// SIMATIC STEP 7 (V5.x) project S_M_Desbobinado
// CPU: CPU312(1)
// station: P_ADR_BUS
// station: Hardware
// station: Equipo SIMATIC 300
// program: Programa S7(1)

SYMBOL_TABLE
"CONTADOR"	C 1	COUNTER
"DESBOBINADO"	FB 1	FB 1	// Función que se encarga del desbobinado
"MULT"	FB 2	FB 2
"MULT_DEBOB"	FB 3	FB 3
"S_CACEROLA"	I 124.0	BOOL
"S_SARTEN"	I 124.1	BOOL
"S_PAELLERA"	I 124.2	BOOL
"S_WOK"	I 124.3	BOOL
"PRESENCIA"	I 124.4	BOOL
"BIT_DE_TRABAJO"	I 124.5	BOOL
"START"	I 124.6	BOOL
"BAJAR_CONT"	I 124.7	BOOL
"SARTEN"	I 125.0	BOOL
"CACEROLA"	I 125.1	BOOL
"WOK"	I 125.2	BOOL
"PAELLERA"	I 125.3	BOOL
"Cycle Execution"	OB 1	OB 1
"C_CACEROLA"	PIW 651	INT
"C_SARTEN"	PIW 653	INT
"C_WOK"	PIW 655	INT
"C_PAELLERA"	PIW 657	INT
"MCENTRO"	PIW 659	INT
"PLANCHAS"	PIW 661	WORD
"ABRIRMCENTRO"	Q 100.0	BOOL
"DESBOBINAR"	Q 100.1	BOOL
"BIT_OK"	Q 100.2	BOOL
"BIT_ERROR"	Q 100.3	BOOL
"STBY"	Q 100.4	BOOL
"STBY_SARTEN"	Q 101.0	BOOL
"STBY_CACEROLA"	Q 101.1	BOOL
"STBY_PAELLERA"	Q 101.2	BOOL
"STBY_WOK"	Q 101.3	BOOL
END_SYMBOL_TABLE

FUNCTION_BLOCK "DESBOBINADO"	// FB 1
TITLE = DESBOBINADO
VERSION : 0.1
VAR_INPUT
  SENSOR : BOOL ;
  PRESENCIA : BOOL ;
  CENTRO : INT ;
  bit_de_trabajo : BOOL ;
  MCENTRO : INT ;
  Contador : COUNTER ;
  START : BOOL ;
  PLANCHAS : WORD  := W#16#100;
END_VAR
VAR_OUTPUT
  ABRIRMCENTRO : BOOL ;
  DESBOBINAR : BOOL ;
  STBY : BOOL ;
END_VAR
VAR
  x31 : BOOL ;
  x32 : BOOL ;
  x33 : BOOL ;
  x34 : BOOL ;
  s1 : BOOL ;
  FP_Bit_Tr : BOOL ;
  x30 : BOOL ;
  FP_PRESENCIA : BOOL ;
  FP_BDT : BOOL ;
  FP_START : BOOL ;
END_VAR
VAR_TEMP
  watchdog_master : BOOL ;
END_VAR
BEGIN
NETWORK
TITLE = Arranque
      SET;
      A     #bit_de_trabajo;
      FP    #FP_BDT;
      S     #x30;
      R     #x31;
      R     #x32;
      R     #x33;
      R     #x34;
      R     #s1;
NETWORK
TITLE = x31 a x32
//Comparacion medida centro con medida nominal del centro para pasar de x31 a x32
      A     #x31;
      A(;
      L     #CENTRO;
      L     #MCENTRO;
      ==R;
      );
      R     #x31;
      S     #x32;
NETWORK
TITLE = x32 a x33
//Presencia detecta que la plancha esta en posicion para empezar el proceso de 
//desbobinado-cizallado
      A     #x32;
      A     #PRESENCIA;
      FP    #FP_PRESENCIA;
      R     #x32;
      S     #x33;
NETWORK
TITLE = x33 a x34
//Detecta que la plancha esta lista para ser cizallada
      A     #x33;
      A     #SENSOR;
      R     #x33;
      S     #x34;
NETWORK
TITLE = x34 a x33
//si el contador no ha acabado
      A     #x34;
      T     LD 1;
      TAK;
      T     LD 5;
      L     #Contador;
      T     LW 9;
      L     LD 5;
      L     LD 1;
      A     C [LW 9];
      AN    #SENSOR;
      R     #x34;
      S     #x33;
NETWORK
TITLE = x34 a s1
//si el contador ha cabado
      A     #x34;
      T     LD 1;
      TAK;
      T     LD 5;
      L     #Contador;
      T     LW 9;
      L     LD 5;
      L     LD 1;
      AN    C [LW 9];
      AN    #SENSOR;
      AN    #PRESENCIA;
      R     #x34;
      S     #x30;
NETWORK
TITLE = Tratamiento de bit de fin
      A     #x30;
      =     #STBY;
NETWORK
TITLE = Abrir centro
      A     #x31;
      =     #ABRIRMCENTRO;
NETWORK
TITLE = Carga del contador y desbobinado en x32
      A     #x32;
      S     #DESBOBINAR;
      L     #PLANCHAS;
      T     LD 1;
      TAK;
      T     LD 5;
      L     #Contador;
      T     LW 9;
      L     LD 5;
      L     LD 1;
      S     C [LW 9];
NETWORK
TITLE = Resta del contador y salida del x33
      A     #x33;
      S     #DESBOBINAR;
NETWORK
TITLE =
      A     #x34;
      R     #DESBOBINAR;
NETWORK
TITLE = De X30 a X31
      A     #START;
      FP    #FP_START;
      A     #x30;
      R     #x30;
      S     #x31;
END_FUNCTION_BLOCK

FUNCTION_BLOCK "MULT_DEBOB"	// FB 3
VERSION : 0.1
VAR_INPUT
  S_CACEROLA : BOOL ;
  S_SARTEN : BOOL ;
  S_PAELLERA : BOOL ;
  S_WOK : BOOL ;
  PRESENCIA : BOOL ;
  C_CACEROLA : INT ;
  C_SARTEN : INT ;
  C_WOK : INT ;
  C_PAELLERA : INT ;
  BIT_DE_TRABAJO : BOOL ;
  MCENTRO : INT ;
  CONTADOR : COUNTER ;
  PLANCHAS : WORD ;
  SARTEN : BOOL ;
  CACEROLA : BOOL ;
  WOK : BOOL ;
  PAELLERA : BOOL ;
  START : BOOL ;
END_VAR
VAR_OUTPUT
  ABRIRMCENTRO : BOOL ;
  DESBOBINAR : BOOL ;
  BIT_OK : BOOL ;
  BIT_ERROR : BOOL ;
  STBY : BOOL ;
  STBY_SAR : BOOL ;
  STBY_CAC : BOOL ;
  STBY_WOK : BOOL ;
  STBY_PAELL : BOOL ;
END_VAR
VAR
  CAC_DESB : FB 1;
  SART_DESB : FB 1;
  WOK_DESB : FB 1;
  PAELL_DESB : FB 1;
  START_SAR : BOOL ;
  START_CAC : BOOL ;
  START_WOK : BOOL ;
  START_PAELL : BOOL ;
  FP_BDT : BOOL ;
  X1 : BOOL ;
  X2 : BOOL ;
  X3 : BOOL ;
  X4 : BOOL ;
  X5 : BOOL ;
  X6 : BOOL ;
  BDT : BOOL ;
  FP_START : BOOL ;
  FLAG_DESB : BOOL ;
  FP_DESBOB : BOOL ;
  F_START : BOOL ;
END_VAR
BEGIN
NETWORK
TITLE =
      A     #X2;
      JCN   _008;
      S     #BDT;
      BLD   14;
      =     L 6.0;
      L     DINO;
      T     LW 4;
      CDB;
      OPN   DI [LW 4];
      TAR2  LD 0;
      A     DBX [AR2,P#0.1];
      =     #SART_DESB.SENSOR;
      A     DBX [AR2,P#0.4];
      =     #SART_DESB.PRESENCIA;
      L     DBW [AR2,P#4.0];
      T     #SART_DESB.CENTRO;
      A     DBX [AR2,P#95.3];
      =     #SART_DESB.bit_de_trabajo;
      L     DBW [AR2,P#12.0];
      T     #SART_DESB.MCENTRO;
      L     DBW [AR2,P#14.0];
      T     #SART_DESB.Contador;
      A     DBX [AR2,P#94.0];
      =     #SART_DESB.START;
      L     DBW [AR2,P#16.0];
      T     #SART_DESB.PLANCHAS;
      +AR2  P#40.0;
      UC    "DESBOBINADO";
      LAR2  LD 0;
      A     #SART_DESB.ABRIRMCENTRO;
      =     DBX [AR2,P#20.0];
      A     #SART_DESB.DESBOBINAR;
      =     DBX [AR2,P#20.1];
      A     #SART_DESB.STBY;
      =     DBX [AR2,P#20.5];
      CDB;
      BLD   15;
_008: NOP   0;
NETWORK
TITLE =
      A     #X3;
      JCN   _009;
      S     #BDT;
      BLD   14;
      =     L 6.0;
      L     DINO;
      T     LW 4;
      CDB;
      OPN   DI [LW 4];
      TAR2  LD 0;
      A     DBX [AR2,P#0.0];
      =     #CAC_DESB.SENSOR;
      A     DBX [AR2,P#0.4];
      =     #CAC_DESB.PRESENCIA;
      L     DBW [AR2,P#2.0];
      T     #CAC_DESB.CENTRO;
      A     DBX [AR2,P#95.3];
      =     #CAC_DESB.bit_de_trabajo;
      L     DBW [AR2,P#12.0];
      T     #CAC_DESB.MCENTRO;
      L     DBW [AR2,P#14.0];
      T     #CAC_DESB.Contador;
      A     DBX [AR2,P#94.1];
      =     #CAC_DESB.START;
      L     DBW [AR2,P#16.0];
      T     #CAC_DESB.PLANCHAS;
      +AR2  P#22.0;
      UC    "DESBOBINADO";
      LAR2  LD 0;
      A     #CAC_DESB.ABRIRMCENTRO;
      =     DBX [AR2,P#20.0];
      A     #CAC_DESB.DESBOBINAR;
      =     DBX [AR2,P#20.1];
      A     #CAC_DESB.STBY;
      =     DBX [AR2,P#20.6];
      CDB;
      BLD   15;
_009: NOP   0;
NETWORK
TITLE =
      A     #X4;
      JCN   _010;
      S     #BDT;
      BLD   14;
      =     L 6.0;
      L     DINO;
      T     LW 4;
      CDB;
      OPN   DI [LW 4];
      TAR2  LD 0;
      A     DBX [AR2,P#0.3];
      =     #WOK_DESB.SENSOR;
      A     DBX [AR2,P#0.4];
      =     #WOK_DESB.PRESENCIA;
      L     DBW [AR2,P#6.0];
      T     #WOK_DESB.CENTRO;
      A     DBX [AR2,P#95.3];
      =     #WOK_DESB.bit_de_trabajo;
      L     DBW [AR2,P#12.0];
      T     #WOK_DESB.MCENTRO;
      L     DBW [AR2,P#14.0];
      T     #WOK_DESB.Contador;
      A     DBX [AR2,P#94.2];
      =     #WOK_DESB.START;
      L     DBW [AR2,P#16.0];
      T     #WOK_DESB.PLANCHAS;
      +AR2  P#58.0;
      UC    "DESBOBINADO";
      LAR2  LD 0;
      A     #WOK_DESB.ABRIRMCENTRO;
      =     DBX [AR2,P#20.0];
      A     #WOK_DESB.DESBOBINAR;
      =     DBX [AR2,P#20.1];
      A     #WOK_DESB.STBY;
      =     DBX [AR2,P#20.7];
      CDB;
      BLD   15;
_010: NOP   0;
NETWORK
TITLE =
      A     #X5;
      JCN   _011;
      S     #BDT;
      BLD   14;
      =     L 6.0;
      L     DINO;
      T     LW 4;
      CDB;
      OPN   DI [LW 4];
      TAR2  LD 0;
      A     DBX [AR2,P#0.2];
      =     #PAELL_DESB.SENSOR;
      A     DBX [AR2,P#0.4];
      =     #PAELL_DESB.PRESENCIA;
      L     DBW [AR2,P#8.0];
      T     #PAELL_DESB.CENTRO;
      A     DBX [AR2,P#95.3];
      =     #PAELL_DESB.bit_de_trabajo;
      L     DBW [AR2,P#12.0];
      T     #PAELL_DESB.MCENTRO;
      L     DBW [AR2,P#14.0];
      T     #PAELL_DESB.Contador;
      A     DBX [AR2,P#94.3];
      =     #PAELL_DESB.START;
      L     DBW [AR2,P#16.0];
      T     #PAELL_DESB.PLANCHAS;
      +AR2  P#76.0;
      UC    "DESBOBINADO";
      LAR2  LD 0;
      A     #PAELL_DESB.ABRIRMCENTRO;
      =     DBX [AR2,P#20.0];
      A     #PAELL_DESB.DESBOBINAR;
      =     DBX [AR2,P#20.1];
      A     #PAELL_DESB.STBY;
      =     DBX [AR2,P#21.0];
      CDB;
      BLD   15;
_011: NOP   0;
NETWORK
TITLE =
      A     #X2;
      =     #START_SAR;
NETWORK
TITLE =
      A     #X3;
      =     #START_CAC;
NETWORK
TITLE =
      A     #X4;
      =     #START_WOK;
NETWORK
TITLE =
      A     #X5;
      =     #START_PAELL;
NETWORK
TITLE =
      A     #BIT_DE_TRABAJO;
      FP    #FP_BDT;
      R     #START_SAR;
      R     #START_CAC;
      R     #START_WOK;
      R     #START_PAELL;
      S     #X1;
      R     #X2;
      R     #X3;
      R     #X4;
      R     #X5;
      R     #X6;
NETWORK
TITLE =
      A     #START;
      FP    #FP_START;
      =     #F_START;
NETWORK
TITLE =
      A     #F_START;
      A     #X1;
      A     #SARTEN;
      R     #X1;
      S     #X2;
NETWORK
TITLE =
      A     #F_START;
      A     #X1;
      A     #CACEROLA;
      R     #X1;
      S     #X3;
NETWORK
TITLE =
      A     #F_START;
      A     #X1;
      A     #WOK;
      R     #X1;
      S     #X4;
NETWORK
TITLE =
      A     #F_START;
      A     #X1;
      A     #PAELLERA;
      R     #X1;
      S     #X5;
NETWORK
TITLE =
      A     #DESBOBINAR;
      FP    #FP_DESBOB;
      S     #FLAG_DESB;
NETWORK
TITLE =
      A     #X2;
      A     #FLAG_DESB;
      A     #STBY_SAR;
      R     #FLAG_DESB;
      R     #X2;
      S     #X6;
NETWORK
TITLE =
      A     #X3;
      A     #FLAG_DESB;
      A     #STBY_CAC;
      R     #FLAG_DESB;
      R     #X3;
      S     #X6;
NETWORK
TITLE =
      A     #X4;
      A     #FLAG_DESB;
      A     #STBY_WOK;
      R     #FLAG_DESB;
      R     #X4;
      S     #X6;
NETWORK
TITLE =
      A     #X5;
      A     #FLAG_DESB;
      A     #STBY_PAELL;
      R     #FLAG_DESB;
      R     #X5;
      S     #X6;
NETWORK
TITLE =
      A     #X1;
      =     #STBY;
NETWORK
TITLE =
      A     #X6;
      =     #BIT_OK;
END_FUNCTION_BLOCK

DATA_BLOCK DB 1
VERSION : 0.0
"MULT_DEBOB"
BEGIN
END_DATA_BLOCK

ORGANIZATION_BLOCK "Cycle Execution"	// OB 1
TITLE = "Main Program Sweep (Cycle)"
VERSION : 0.1
VAR_TEMP
  OB1_EV_CLASS : BYTE ;	//Bits 0-3 = 1 (Coming event), Bits 4-7 = 1 (Event class 1)
  OB1_SCAN_1 : BYTE ;	//1 (Cold restart scan 1 of OB 1), 3 (Scan 2-n of OB 1)
  OB1_PRIORITY : BYTE ;	//Priority of OB Execution
  OB1_OB_NUMBR : BYTE ;	//1 (Organization block 1, OB1)
  OB1_RESERVED_1 : BYTE ;	//Reserved for system
  OB1_RESERVED_2 : BYTE ;	//Reserved for system
  OB1_PREV_CYCLE : INT ;	//Cycle time of previous OB1 scan (milliseconds)
  OB1_MIN_CYCLE : INT ;	//Minimum cycle time of OB1 (milliseconds)
  OB1_MAX_CYCLE : INT ;	//Maximum cycle time of OB1 (milliseconds)
  OB1_DATE_TIME : DATE_AND_TIME ;	//Date and time OB1 started
END_VAR
BEGIN
NETWORK
TITLE =
      SET;
      CALL  "MULT_DEBOB" , DB 1 (
           S_CACEROLA               := "S_CACEROLA",
           S_SARTEN                 := "S_SARTEN",
           S_PAELLERA               := "S_PAELLERA",
           S_WOK                    := "S_WOK",
           PRESENCIA                := "PRESENCIA",
           C_CACEROLA               := "C_CACEROLA",
           C_SARTEN                 := "C_SARTEN",
           C_WOK                    := "C_WOK",
           C_PAELLERA               := "C_PAELLERA",
           BIT_DE_TRABAJO           := "BIT_DE_TRABAJO",
           MCENTRO                  := "MCENTRO",
           CONTADOR                 := "CONTADOR",
           PLANCHAS                 := "PLANCHAS",
           SARTEN                   := "SARTEN",
           CACEROLA                 := "CACEROLA",
           WOK                      := "WOK",
           PAELLERA                 := "PAELLERA",
           START                    := "START",
           ABRIRMCENTRO             := "ABRIRMCENTRO",
           DESBOBINAR               := "DESBOBINAR",
           BIT_OK                   := "BIT_OK",
           BIT_ERROR                := "BIT_ERROR",
           STBY                     := "STBY",
           STBY_SAR                 := "STBY_SARTEN",
           STBY_CAC                 := "STBY_CACEROLA",
           STBY_WOK                 := "STBY_WOK",
           STBY_PAELL               := "STBY_PAELLERA");
NETWORK
TITLE =
      A     "BAJAR_CONT";
      CD    "CONTADOR";
END_ORGANIZATION_BLOCK
